{attribute addProperty BoxType "EJ7211-0011-0026"}
{attribute addProperty Id "Position_actual_valueAT %I*UDINT324"}
{attribute addProperty CRC "219267348"}
{attribute addProperty SizeInBites "32"}
{attribute addProperty SizeInBytes "4"}
TYPE DS402_Position_actual_value_0D11C114 :
STRUCT
	{attribute addProperty Name "Position_actual_value"}
	Position_actual_value AT %I* : UDINT;
END_STRUCT
END_TYPE

(* stored: Version 1.2.0.0, ProductVersion 3.1.4024.9
   DUT DS402_Position_actual_value_0D11C114: Id {99915269-ab36-4524-bd23-3eef17955ecf} *)
